(*
Nazwa:			E_DragStationState
Opis:			Stan stacji przeciągania pneumatyczengo
Wersja:			v0.2
Data:			2022-05-18
Autor:			DJ
Urzadzenia:		Przeciąganie butelek
Konfiguracja:	
Info:
*)


TYPE E_DragStationStatePneum :
(
	eDisabled					:= 0,  			//Wyłączona
	eReady						:= 2,				//Gotowość
	ePreparingToMove			:= 4,	//Przygotowanie do ruchu
	eLifting					:= 7, 			//Podnoszenie
	ePrepareToDrag				:= 8, 		//Przygotowanie do przeicagana
	eDraging					:= 9,			//Przeciaganie
	eDragingDone				:= 10,
	eEndingOfDrag				:= 11,
	eEndingOfDragDone			:= 12,
	eLowering					:= 13,			//Opuszczanie 
	eDraged						:= 14,  			//Powrót do bazy, przeciągnięte
	eDragedDone					:= 15
):=eDisabled;

END_TYPE

(* stored: Version 1.1.0.1, ProductVersion 3.1.4026.13, FileIdentifier 29c4c6efdf852b321af2da46e88747fee0d7bdc9, FileSignature 9bd64552a5f686b760c9fb1873c194e49bc7815f6390f639ebbecd21836a825d81cebb1bf76d0f333b043d28040e9261d9cda956b6d8fc3817d8d9fb15bbcf1d1fa8965e85d440aa44e17448d9e77d1fb1eb97b553673ce81e3a95aaf7f7aeea02795dd1003615833eb9b02610cd46a74058958e7a5513604c06166f347ed454fd976aa7449e10981cb1b196a479833c3608fd3b571951d4604378033e919fc23922a748f96fe4ef36d4cc8b9f5699d2c2954b54b8fd35562a3ab3a63eb3bbfe666abecfd66ea5cfa954cbe9728dde98e1144ca143b2d90ac0e915c3093645bed95081e4d4185c438c83997cdc3ca93da9796dd3413dd68884ab09b88440032c
   DUT E_DragStationStatePneum: Id {ab97ea73-441f-4bca-9fb2-5cb411c072a6} *)
